(* Logix 5000 project; controller miPrimerPrograma Emulate 5570 rev 32.11; software revision 32.02 *)

TASK T00_MainTask (continuous, watchdog 500 ms) : P00_MainProgram

MODULES
   Local : Emulate 5570 (ICP 2, rev 32.11)
END_MODULES

VAR_GLOBAL   (* controller tags *)
   botonArranque : BOOL;
   botonParo : BOOL;
   entrada1 : BOOL := 1;   // memoriaVirtual
   entrada2 : BOOL := 1;   // memoriaVirtual
   motor : BOOL;
   salida1 : BOOL := 1;   // memoriaVirual
END_VAR

PROGRAM P00_MainProgram   (* main routine R00_MainRoutine *)
VAR
   ALM_01 : ALARM;
   Counters : COUNTER[25] := ([0].PRE := 10, [1].PRE := 10, [1].ACC := 315, [1].DN := 1);
   habilitarTimmer : BOOL;
   motor2 : BOOL;
   ONS : BOOL[32];
   salida2 : BOOL := 1;
   Timmer : TIMER[25] := ([0].PRE := 5000, [1].PRE := 5000, [2].PRE := 3000, [3].PRE := 1000, [3].ACC := 868, [3].EN := 1, [3].TT := 1, [4].PRE := 15000, [4].ACC := 15014);
END_VAR

ROUTINE R00_MainRoutine   (* ladder *)
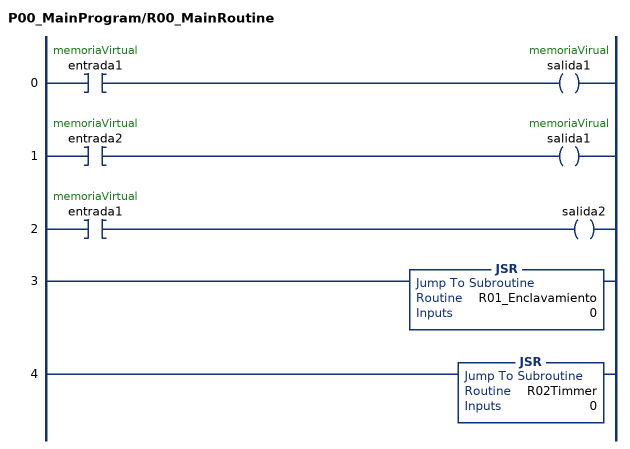
   0: XIC(entrada1)OTE(salida1);
   1: XIC(entrada2)OTE(salida1);
   2: XIC(entrada1)OTE(salida2);
   3: JSR(R01_Enclavamiento,0);
   4: JSR(R02Timmer,0);
END_ROUTINE

ROUTINE R01_Enclavamiento   (* ladder *)
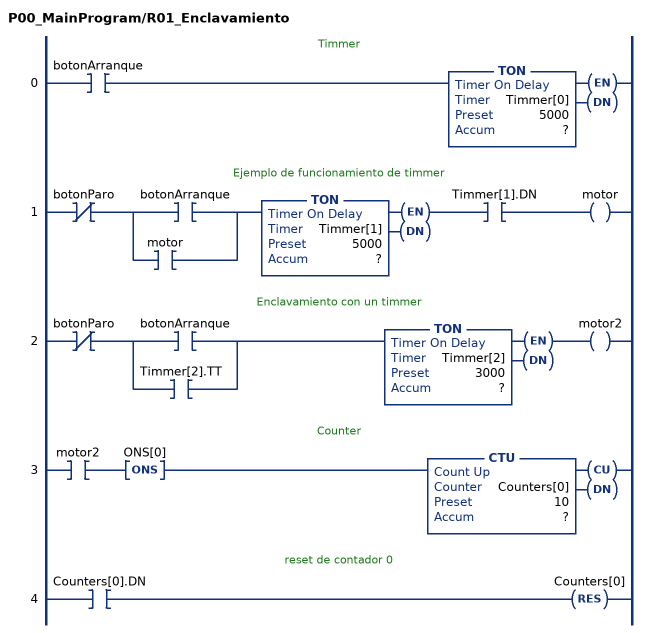
   // Timmer
   0: XIC(botonArranque)TON(Timmer[0],?,?);
   // Ejemplo de funcionamiento de timmer
   1: XIO(botonParo)[XIC(botonArranque) ,XIC(motor) ]TON(Timmer[1],?,?)XIC(Timmer[1].DN)OTE(motor);
   // Enclavamiento con un timmer
   2: XIO(botonParo)[XIC(botonArranque) ,XIC(Timmer[2].TT) ]TON(Timmer[2],?,?)OTE(motor2);
   // Counter
   3: XIC(motor2)ONS(ONS[0])CTU(Counters[0],?,?);
   // reset de contador 0
   4: XIC(Counters[0].DN)RES(Counters[0]);
END_ROUTINE

ROUTINE R02Timmer   (* ladder *)
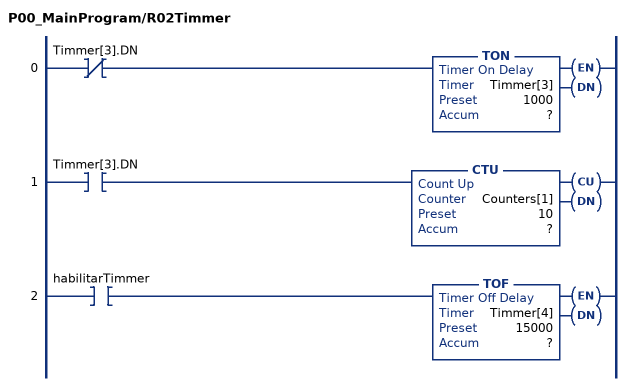
   0: XIO(Timmer[3].DN)TON(Timmer[3],?,?);
   1: XIC(Timmer[3].DN)CTU(Counters[1],?,?);
   2: XIC(habilitarTimmer)TOF(Timmer[4],?,?);
END_ROUTINE
END_PROGRAM
